TEXTLIST AxesDialogDeltaUnitsTextList
  0 = 'd / m / s'
  1 = 'degrees'
  2 = 'radians'
   = ''
END_TEXTLIST

(* stored: Version 1.1.0.1, ProductVersion 3.1.4018.5
   TextList AxesDialogDeltaUnitsTextList: Id {121db9de-1d6d-4973-b33d-4bf4d2666712} *)
